// TIA Portal V17 export
// export: Created 2022-03-12T16:05:15.7862598Z, ExportSetting WithDefaults, DisplayName Totally Integrated Automation Portal, DisplayVersion V17, DisplayName TIA Portal Openness, DisplayVersion V17, DisplayName TIA Portal Version Control Interface, DisplayVersion V17, DisplayName STEP 7 Professional, DisplayVersion V17, DisplayName STEP 7 Safety, DisplayVersion V17, DisplayName WinCC Advanced / Unified PC, DisplayVersion V17
DATA_BLOCK "InstUN_00_Main"   // DB31620
TITLE = instUN00_00_Main
AUTHOR : tech.team.motioncontrol@siemens.com
FAMILY : CPG
VERSION : 1.0
// Support: tech.team.motioncontrol@siemens.com
// Fax: +49 (0) 9131/98-1297
// stored: AutoNumber true, DBAccessibleFromOPCUA true, DBAccessibleFromWebserver true, InstanceOfName UN_00_Main, InstanceOfType FB
"UN_00_Main"
   // VAR
   //    instPackML_ModuleSum { ExternalAccessible := 'False'; ExternalVisible := 'False'; ExternalWritable := 'False'; S7_SetPoint := 'True'} : "UN_01_PackML_ModuleSum";
   //    instPackML { ExternalAccessible := 'False'; ExternalVisible := 'False'; ExternalWritable := 'False'; S7_SetPoint := 'True'} : "UN_02_PackML";
   //    instLineComm { ExternalAccessible := 'False'; ExternalVisible := 'False'; ExternalWritable := 'False'; S7_SetPoint := 'True'} : "UN_03_LineComm";
   //    instEventControl { ExternalAccessible := 'False'; ExternalVisible := 'False'; ExternalWritable := 'False'; S7_SetPoint := 'True'} : "UN_04_EventControl";
   //    instEventSummation { ExternalAccessible := 'False'; ExternalVisible := 'False'; ExternalWritable := 'False'; S7_SetPoint := 'True'} : "UN_05_EventSummation";
   //    instMiscFunctions { ExternalAccessible := 'False'; ExternalVisible := 'False'; ExternalWritable := 'False'; S7_SetPoint := 'True'} : "UN_06_MiscFunctions";
   //    instRecipeControl { ExternalAccessible := 'False'; ExternalVisible := 'False'; ExternalWritable := 'False'; S7_SetPoint := 'True'} : "UN_07_RecipeControl";
   // END_VAR
BEGIN
END_DATA_BLOCK
